# EPICS substitutions: apps/caenHvApp/Db/sums/HVDCb_sums.substitutions
file "db/HVDC_sums.db" {
    pattern {S,R,L}
    {"3","1","1"}
    {"3","1","2"}
    {"3","2","3"}
    {"3","2","4"}
    {"3","3","5"}
    {"3","3","6"}
    {"4","1","1"}
    {"4","1","2"}
    {"4","2","3"}
    {"4","2","4"}
    {"4","3","5"}
    {"4","3","6"}
    {"5","1","1"}
    {"5","1","2"}
    {"5","2","3"}
    {"5","2","4"}
    {"5","3","5"}
    {"5","3","6"}
}
